# EPICS SNL sequencer program: siteApps/SCL3Cooldown-sim-2-O/cooldownApp/src/CDOM143.stt
program CDOM143Logic
option +r;

%% #include <math.h>

int om143LogicProc[1];
assign om143LogicProc to {
":CDLogic.PROC"
};
monitor om143LogicProc;

float valveVal[1];
assign valveVal to {
":Valve"
};

monitor valveVal;

evflag  evFanout;
sync	valveVal	evFanout;

int index = 0;
assign index to "SCL3:CD-OM143:IndexPV";
monitor index;

int proc = 1;

float om143Val;
assign om143Val to "SCL3:CD-OM143:Value";
monitor om143Val;

float cdDelay;
assign cdDelay to "SCL3:CD-OM143:ScanTime";
monitor cdDelay;

float	valvewave[1];
assign	valvewave to "SCL3:CD-OM143:ValveWave";
monitor valvewave;

ss ssCDOM143
{
	state CDOM143
	{
		when(delay(cdDelay))
		{
			if(index == 0  || index == 1  || index == 8  || index == 10 ||
			   index == 12 || index == 14 || index == 16 || index == 18 || index == 20 ||
			   index == 22 || index == 24 || index == 26 || index == 28 || index == 30 ||
			   index == 32 || index == 34 || index == 36 || index == 38 || index == 40 ||
			   index == 42 || index == 44 || index == 46 || index == 48 || index == 50 ||
			   index == 52 || index == 54 || index == 56 || index == 58 || index == 60 ||
			   index == 62 || index == 64 || index == 66 || index == 68 || index == 70 ||
			   index == 72 || index == 75 || index == 78 || index == 81 || index == 84 ||
			   index == 87 || index == 90 || index == 93 || index == 96 || index == 99 ||
			   index == 102|| index == 105)
			{
				if(om143Val == 1) {
					om143Val = 0;
					index++;
					pvPut(index, SYNC);
				} else {
					om143Val = valveVal[index];
				};
			}
			else
			{
				if(om143Val == 100) {
					om143Val = 0;
					index++;
					pvPut(index, SYNC);
				} else {
					om143Val = valveVal[index];
				};
			};

			pvPut(om143Val, SYNC);
			if(index < 107)
			{
				om143LogicProc[index] = proc;
				pvPut(om143LogicProc[index], SYNC);
			};
		}state CDOM143
	}

}

ss ssOM143ValveWave
{
	state init
	{
		when(TRUE)
		{
			efClear(evFanout);
		}state MakeOM143ValveWave
	}

	state MakeOM143ValveWave
	{
		when(efTestAndClear(evFanout))
		{
			int idx = 0;
			%%for(idx = 0; idx < 107;idx++)
				valvewave[idx] = valveVal[idx];

			pvPut(valvewave, SYNC);
		}state MakeOM143ValveWave
	}
}
